FUNCTION_BLOCK FB_LightController
VAR
	_iLight									: I_LightBase;
	_iLightB								: I_LightDimmable;
	                    	    			
	fbLightGroup							: FB_LightGroup;
	
	nBrightness								: USINT := 100;
	                    	    			
	bToggle									: BOOL;
	bSwitch									: BOOL;
	bSetBrightness							: BOOL;
	                    	    			
	tToggle									: R_TRIG;
	tSwitchON								: R_TRIG;
	tSwitchOFF								: F_TRIG;
	tSetBrightness							: R_TRIG;
	                    	    			
	bGroupSwitch							: BOOL;
	bSetGroupBrightness						: BOOL;
	                    	    			
	tGroupSwitchON							: R_TRIG;
	tGroupSwitchOFF							: F_TRIG;
	tSetGroupBrightness						: R_TRIG;
	                    	    			
	eSwitchOptions							: (WAIT, TOGGLE, SWITCHON, SWITCHOFF, SETBRIGHTNESS, GROUPSWITCHON, GROUPSWITCHOFF, SETGROUPBRIGHTNESS);
	
	eSwitchControlledLightObjectByLightID	: (LIGHT_ONE, LIGHT_TWO, LIGHT_THREE, LIGHT_FOUR, LIGHT_FIVE, LIGHT_SIX, LIGHT_SEVEN, LIGHT_EIGHT);
	nSwitchControlledLightObjectByLightID	: USINT;
	
	aOriginalInstanceOfLightFB				: ARRAY[0..MAIN.NUMBER_OF_REG_LIGHTS-1] OF FB_LightBase;
	aOriginalInstanceOfDimmableLightFB		: ARRAY[0..MAIN.NUMBER_OF_DIMMABLE_LIGHTS-1] OF FB_LightBase;

END_VAR

fbLightGroup();

CASE eSwitchOptions OF
	WAIT:
		//do nothing
	TOGGLE:
		_iLight.Toggle();
		eSwitchOptions := WAIT;
	SWITCHON:
		_iLight.TurnON();
		eSwitchOptions := WAIT;
	SWITCHOFF:
		_iLight.TurnOFF();
		eSwitchOptions := WAIT;
	SETBRIGHTNESS:
		IF __QUERYINTERFACE(_iLight, _iLightB) THEN
			_iLightB.Brightness := nBrightness;	
		END_IF
		eSwitchOptions := WAIT;
	GROUPSWITCHON:
		fbLightGroup.TurnON();
		eSwitchOptions := WAIT;
	GROUPSWITCHOFF:
		fbLightGroup.TurnOFF();
		eSwitchOptions := WAIT;
	SETGROUPBRIGHTNESS:
		fbLightGroup.SetBrightness(nBrightness);
		eSwitchOptions := WAIT;
END_CASE

CASE eSwitchControlledLightObjectByLightID OF
	LIGHT_ONE:
		nSwitchControlledLightObjectByLightID := 1;
	LIGHT_TWO:
		nSwitchControlledLightObjectByLightID := 2;
	LIGHT_THREE:
		nSwitchControlledLightObjectByLightID := 3;
	LIGHT_FOUR:
		nSwitchControlledLightObjectByLightID := 4;
	LIGHT_FIVE:
		nSwitchControlledLightObjectByLightID := 5;
	LIGHT_SIX:
		nSwitchControlledLightObjectByLightID := 6;
	LIGHT_SEVEN:
		nSwitchControlledLightObjectByLightID := 7;
	LIGHT_EIGHT:
		nSwitchControlledLightObjectByLightID := 8;
END_CASE

IF nSwitchControlledLightObjectByLightID <= MAIN.NUMBER_OF_REG_LIGHTS THEN
	ipLight := aOriginalInstanceOfLightFB[nSwitchControlledLightObjectByLightID-1];
ELSIF nSwitchControlledLightObjectByLightID > MAIN.NUMBER_OF_REG_LIGHTS THEN
	ipLight := aOriginalInstanceOfDimmableLightFB[nSwitchControlledLightObjectByLightID-MAIN.NUMBER_OF_REG_LIGHTS-1];
ELSIF nSwitchControlledLightObjectByLightID > MAIN.MAXIMUM_NUMBER_OF_LIGHTS THEN
	ipLight := aOriginalInstanceOfDimmableLightFB[MAIN.MAXIMUM_NUMBER_OF_LIGHTS-1];
END_IF


tToggle(CLK := bToggle);
tSwitchON(CLK := bSwitch);
tSwitchOFF(CLK := bSwitch);
tSetBrightness(CLK := bSetBrightness);

tGroupSwitchOFF(CLK := bGroupSwitch);
tGroupSwitchON(CLK := bGroupSwitch);
tSetGroupBrightness(CLK := bSetGroupBrightness);

IF tToggle.Q THEN
	eSwitchOptions := TOGGLE;
	bToggle := FALSE;									
END_IF

IF tSwitchON.Q THEN
	eSwitchOptions := SWITCHON;
END_IF

IF tSwitchOFF.Q THEN
	eSwitchOptions := SWITCHOFF;
END_IF

IF tSetBrightness.Q THEN
	eSwitchOptions := SETBRIGHTNESS;
	bSetBrightness := FALSE;
END_IF

IF tGroupSwitchON.Q THEN
	eSwitchOptions := GROUPSWITCHON;
END_IF

IF tGroupSwitchOFF.Q THEN
	eSwitchOptions := GROUPSWITCHOFF;
END_IF

IF tSetGroupBrightness.Q THEN
	eSwitchOptions := SETGROUPBRIGHTNESS;
	bSetGroupBrightness := FALSE;
END_IF

METHOD FB_init : BOOL
VAR_INPUT
	bInitRetains	: BOOL; // if TRUE, the retain variables are initialized (warm start / cold start)
	bInCopyCode		: BOOL;  // if TRUE, the instance afterwards gets moved into the copy code (online change)
END_VAR
VAR
	nCounter: INT;
END_VAR
_iLight := aOriginalInstanceOfLightFB[0];

FOR nCounter := 0 TO MAIN.NUMBER_OF_REG_LIGHTS-1 DO
fbLightGroup.ImportLight(aOriginalInstanceOfLightFB[nCounter]);
END_FOR

FOR nCounter := 0 TO MAIN.NUMBER_OF_DIMMABLE_LIGHTS-1 DO
fbLightGroup.ImportLight(aOriginalInstanceOfDimmableLightFB[nCounter]);
END_FOR
END_METHOD

PROPERTY ipLight : I_LightBase
GET
ipLight := _iLight;
END_GET
SET
_iLight := ipLight;
END_SET
END_PROPERTY

END_FUNCTION_BLOCK

(* stored: Version 1.1.0.1, ProductVersion 3.1.4024.12
   POU FB_LightController: Id {9da3a0db-3198-4dea-825b-a1e081e7674e}, SpecialFunc None
   Method FB_init: Id {b012ca00-77bf-49e0-b6a1-96f66c4d5657}
   Property ipLight: Id {ec405ff9-3dab-4d63-9f5a-8feda15492ff}
   Get Get: Id {0ffc156d-193d-45e5-b922-0cc8c69053fe}
   Set Set: Id {2c898839-6876-40e2-8be5-95ed55e6501b} *)
